FUNCTION_BLOCK PUBLIC OB_StopRobotClearStation
VAR_INPUT
END_VAR
VAR_OUTPUT
END_VAR
VAR
	xTrigger :BOOL := FALSE; // triggers processing
	State : eOB_StopRobotClearStaState := eOB_StopRobotClearStaState.eUnknown;
	NextState : eOB_StopRobotClearStaState := eOB_StopRobotClearStaState.eUnknown;
	bFirst : BOOL := TRUE;
	VUT : BYTE; //VehicleID Under Station
	DwellTimer : TON;
	MoveVehicleToLoad: BOOL := TRUE; //We have to send the Vehicle to Load Position # 4 at startup
END_VAR

CASE State OF

eOB_StopRobotClearStaState.eUnknown:
	NextState := eOB_StopRobotClearStaState.eReady;

eOB_StopRobotClearStaState.eInit:

eOB_StopRobotClearStaState.eHoming:

eOB_StopRobotClearStaState.eReady:
IF (xTrigger) THEN
		NextState := eOB_StopRobotClearStaState.eProcessing;
		
		DwellTimer(IN:=FALSE);
	END_IF

eOB_StopRobotClearStaState.eDwell:

eOB_StopRobotClearStaState.eProcessing:
  IF (MoveVehicleToLoad) THEN
	  NextState := eOB_StopRobotClearStaState.eDepart;
  END_IF

eOB_StopRobotClearStaState.eDepart:
	
    Stations.fbRoutePlanner.M_NotifyVehStaCmpl(StationIndex:= MM_CONST.OB_STOP_ROBOT_CLEAR_STA, VehicleID := VUT);
	xTrigger := FALSE;
	MoveVehicleToLoad := FALSE;	
	NextState := eOB_StopRobotClearStaState.eReady;

eOB_StopRobotClearStaState.eError:

ELSE;

END_CASE

IF (State <> NextState) THEN
	bFirst := TRUE;
ELSE
	bFirst := FALSE;
END_IF

State := NextState;

Status.StationsState[MM_CONST.OB_STOP_ROBOT_CLEAR_STA_HMI_STATE] := State;

METHOD PUBLIC ClearVehicleTrigger : BOOL
VAR_INPUT
END_VAR
xTrigger := FALSE;
State := eOB_StopRobotClearStaState.eUnknown;
NextState:= eOB_StopRobotClearStaState.eUnknown;
bFirst  := TRUE;
MoveVehicleToLoad := TRUE; //We have to send the Vehicle to Load Position # 4 at startup
END_METHOD

PROPERTY PUBLIC MoveToLoading : BOOL
SET
MoveVehicleToLoad := MoveToLoading;
END_SET
END_PROPERTY

PROPERTY PUBLIC Trigger : BOOL
SET
xTrigger := Trigger;
END_SET
END_PROPERTY

PROPERTY PUBLIC VehicleUnderTest : BYTE
GET
VehicleUnderTest := VUT;
END_GET
SET
VUT := VehicleUnderTest;
END_SET
END_PROPERTY

END_FUNCTION_BLOCK

(* stored: Version 1.1.0.1, ProductVersion 3.1.4020.12
   POU OB_StopRobotClearStation: Id {4ebeb43e-907a-4019-a0a5-420aa63a9667}, SpecialFunc None
   Method ClearVehicleTrigger: Id {b7098c1e-d1fc-4ec2-b1df-66639cd9ffc3}
   Property MoveToLoading: Id {4c7ea59a-bcb3-415c-9007-8fe1c9cfecd1}
   Set Set: Id {b9674ea6-1294-4251-8340-cb830ed9ebd0}
   Property Trigger: Id {379d2162-3f8a-4e6c-b755-88309af6de26}
   Set Set: Id {e2b351f4-7441-4b22-affb-367fa2ee7e6d}
   Property VehicleUnderTest: Id {99345c28-8d08-4f0c-8947-2857472d7424}
   Get Get: Id {54810044-f560-48ae-87b8-a29789f67911}
   Set Set: Id {32ebcb68-1970-4183-8d7e-d5dcfecd041f} *)
